// TIA Portal V19 export
FUNCTION_BLOCK "TYPIC_C402_IF_SBO1"   // FB111, FBD
TITLE = TYPIC_C402_IF_SBO: Afsluitboom
{ S7_Optimized_Access := 'TRUE' }
AUTHOR : OCOTECH
FAMILY : Typical
NAME : C402.704
// Logisch Object Besturing: C402.704
// 
// 								De interne functie afsluitboom verzorgt de interne besturing,
// 								bewaking en fysieke aansturing van een afsluitboom.
// 
// 								Het akoestisch signaal en de optische signalen behorend bij de
// 								afsluitboom, wordt eveneens via deze functie aangestuurd.
// stored: MemoryReserve 10, SetENOAutomatically false
   VAR_INPUT
      EXT_AUT { ExternalAccessible := 'False'; ExternalVisible := 'False'; ExternalWritable := 'False'} : Bool;   // Externe (hoofd) beveiliging (1 = OK)
      EXT_HW { ExternalAccessible := 'False'; ExternalVisible := 'False'; ExternalWritable := 'False'} : Bool;   // Sturings hardware (PLC) bewaking (1 = OK)
      HULP_KNIP { ExternalAccessible := 'False'; ExternalVisible := 'False'; ExternalWritable := 'False'} : Bool;   // Knippersignaal, x tijd hoog, x tijd laag
      IN_AUT { ExternalAccessible := 'False'; ExternalVisible := 'False'; ExternalWritable := 'False'} : Bool;   // Motorbeveiliging (1 = OK / 0 = storing)
      IN_OPEN { ExternalAccessible := 'False'; ExternalVisible := 'False'; ExternalWritable := 'False'} : Bool;   // Terugmelding: afsluitboom is open
      IN_TOE { ExternalAccessible := 'False'; ExternalVisible := 'False'; ExternalWritable := 'False'} : Bool;   // Terugmelding: afsluitboom is toe
      IN_STO { ExternalAccessible := 'False'; ExternalVisible := 'False'; ExternalWritable := 'False'} : Bool;   // Terugmelding: afsluitboom is buiten dienst
      IN_SCW { ExternalAccessible := 'False'; ExternalVisible := 'False'; ExternalWritable := 'False'} : Bool;   // Werkschakelaar (1 = AAN)
      IN_HND { ExternalAccessible := 'False'; ExternalVisible := 'False'; ExternalWritable := 'False'} : Bool;   // Mechanische handmatige bediening (0 = Hand)
      IN_LVE1_STO { ExternalAccessible := 'False'; ExternalVisible := 'False'; ExternalWritable := 'False'} : Bool;   // Detector lus 1 (1 = OK / 0 = storing)
      IN_LVE2_STO { ExternalAccessible := 'False'; ExternalVisible := 'False'; ExternalWritable := 'False'} : Bool;   // Detector lus 2 (1 = OK / 0 = storing)
      IN_LVE3_STO { ExternalAccessible := 'False'; ExternalVisible := 'False'; ExternalWritable := 'False'} : Bool;   // Detector lus 3 (1 = OK / 0 = storing)
      IN_LVE4_STO { ExternalAccessible := 'False'; ExternalVisible := 'False'; ExternalWritable := 'False'} : Bool;   // Detector lus 4 (1 = OK / 0 = storing)
      IN_LUS1_STS { ExternalAccessible := 'False'; ExternalVisible := 'False'; ExternalWritable := 'False'} : Bool;   // Detectie voertuig door lus 1 (1 = Geen detectie)
      IN_LUS2_STS { ExternalAccessible := 'False'; ExternalVisible := 'False'; ExternalWritable := 'False'} : Bool;   // Detectie voertuig door lus 2 (1 = Geen detectie)
      IN_LUS3_STS { ExternalAccessible := 'False'; ExternalVisible := 'False'; ExternalWritable := 'False'} : Bool;   // Detectie voertuig door lus 3 (1 = Geen detectie)
      IN_LUS4_STS { ExternalAccessible := 'False'; ExternalVisible := 'False'; ExternalWritable := 'False'} : Bool;   // Detectie voertuig door lus 4 (1 = Geen detectie)
      IN_AUT_C402 { ExternalAccessible := 'False'; ExternalVisible := 'False'; ExternalWritable := 'False'} : Bool;   // Beveiligingen: serie geschakelde terugmelding (1 = OK)
      IN_DKN_OPEN { ExternalAccessible := 'False'; ExternalVisible := 'False'; ExternalWritable := 'False'} : Bool;   // 1 = Drukknop ingedrukt, bediening openen
      IN_DKN_TOE { ExternalAccessible := 'False'; ExternalVisible := 'False'; ExternalWritable := 'False'} : Bool;   // 1 = Drukknop ingedrukt, bediening sluiten
      IN_DKN_STOP { ExternalAccessible := 'False'; ExternalVisible := 'False'; ExternalWritable := 'False'} : Bool;   // 1 = Drukknop ingedrukt, bediening stop
      CFG_TYD_STS { ExternalAccessible := 'False'; ExternalVisible := 'False'; ExternalWritable := 'False'} : Time;   // Vertragingstijd storing terugmelding stand bereikt
      CFG_ITYD_POS { ExternalAccessible := 'False'; ExternalVisible := 'False'; ExternalWritable := 'False'} : Time;   // Inschakelvertraging storing eindpositie terugmelding weggevallen
      CFG_UTYD_POS { ExternalAccessible := 'False'; ExternalVisible := 'False'; ExternalWritable := 'False'} : Time;   // Uitschakelvertraging storing eindpositie terugmelding weggevallen
      CFG_ITYD_OAS_SNEL { ExternalAccessible := 'False'; ExternalVisible := 'False'; ExternalWritable := 'False'} : Time;   // Vertragingstijd versneld sluiten afsluitboom na akoestisch en optisch signaal
      CFG_ITYD_OAS { ExternalAccessible := 'False'; ExternalVisible := 'False'; ExternalWritable := 'False'} : Time;   // Vertragingstijd sluiten/openen afsluitboom regulier na akoestisch en optisch signaal
      CFG_UTYD_OAS { ExternalAccessible := 'False'; ExternalVisible := 'False'; ExternalWritable := 'False'} : Time;   // Vertragingstijd uitschakelen akoestische en optische signalen
      CFG_UTYD_MOT { ExternalAccessible := 'False'; ExternalVisible := 'False'; ExternalWritable := 'False'} : Time;   // Vertragingstijd uitschakelen motor na bereiken eindpositie
      CFG_VGV_OPEN { ExternalAccessible := 'False'; ExternalVisible := 'False'; ExternalWritable := 'False'} : Bool;   // 1 = Slagboom moet openen bij bediening openen door hulpdiensten
   END_VAR
   VAR_OUTPUT
      VAR_IF_SBO { ExternalAccessible := 'False'; ExternalVisible := 'False'; ExternalWritable := 'False'} : "C402_VAR_IF_SBO_TYPIC";   // Struct met alle variabelen naar bovenliggende functies
      OUT_OPEN { ExternalAccessible := 'False'; ExternalVisible := 'False'; ExternalWritable := 'False'} : Bool;   // Aansturing openen
      OUT_TOE { ExternalAccessible := 'False'; ExternalVisible := 'False'; ExternalWritable := 'False'} : Bool;   // Aansturing sluiten
      OUT_AKS { ExternalAccessible := 'False'; ExternalVisible := 'False'; ExternalWritable := 'False'} : Bool;   // Aansturen akoestische signalering
      OUT_OPS { ExternalAccessible := 'False'; ExternalVisible := 'False'; ExternalWritable := 'False'} : Bool;   // Aansturen optische signalering
   END_VAR
   VAR_IN_OUT
      STU_IF_SBO : "C402_STU_IF_SBO_TYPIC";   // Struct met alle sturingen naar de functie (IF) in de interne sturing van de afsluitboom
      STU_AFS_IF_SBO : "C402_STU_AFS_IF_SBO_TYPIC";   // Struct met alle sturingen vanuit de interne functie Afsluitsysteem naar de functies (IF) van de afsluitbomen
   END_VAR
   VAR
      STO { ExternalWritable := 'False'} : Struct   // Storingen
         A001 { ExternalAccessible := 'False'; ExternalVisible := 'False'} : Bool;   // Beveiliging aangesproken
         A002 { ExternalAccessible := 'False'; ExternalVisible := 'False'} : Bool;   // Storing van de detector van lus 1
         A003 { ExternalAccessible := 'False'; ExternalVisible := 'False'} : Bool;   // Storing van de detector van lus 2
         A004 { ExternalAccessible := 'False'; ExternalVisible := 'False'} : Bool;   // Storing van de detector van lus 3
         A005 { ExternalAccessible := 'False'; ExternalVisible := 'False'} : Bool;   // Storing van de detector van lus 4
         A006 { ExternalAccessible := 'False'; ExternalVisible := 'False'} : Bool;   // Storing van de motorsturing
         A007 { ExternalAccessible := 'False'; ExternalVisible := 'False'} : Bool;   // Storing motorbeveiliging
         AT01 { ExternalAccessible := 'False'; ExternalVisible := 'False'} : Bool;   // Terugmelding Open niet tijdig bereikt
         AT02 { ExternalAccessible := 'False'; ExternalVisible := 'False'} : Bool;   // Terugmelding Dicht niet tijdig bereikt
         AT03 { ExternalAccessible := 'False'; ExternalVisible := 'False'} : Bool;   // Terugmeldingen Open en Dicht tegelijkertijd
         AT04 { ExternalAccessible := 'False'; ExternalVisible := 'False'} : Bool;   // Terugmelding Open weggevallen
         AT05 { ExternalAccessible := 'False'; ExternalVisible := 'False'} : Bool;   // Terugmelding Dicht weggevallen
         M001 { ExternalAccessible := 'False'; ExternalVisible := 'False'} : Bool;   // Werkschakelaar uitgeschakeld
         M002 { ExternalAccessible := 'False'; ExternalVisible := 'False'} : Bool;   // Mechanische handbediening uitgenomen
      END_STRUCT;
      VAR { ExternalWritable := 'False'} : Struct   // Variabelen
         CMD_AKS { ExternalAccessible := 'False'; ExternalVisible := 'False'} : Bool;   // Aansturen akoestische signalering
         CMD_OPS { ExternalAccessible := 'False'; ExternalVisible := 'False'} : Bool;   // Aansturen optische signalering
         VWA_AT04 { ExternalAccessible := 'False'; ExternalVisible := 'False'} : Bool;   // Voorwaarden voldaan voor storing AT04
         VWA_AT05 { ExternalAccessible := 'False'; ExternalVisible := 'False'} : Bool;   // Voorwaarden voldaan voor storing AT05
         MOT_STS_AAN { ExternalAccessible := 'False'; ExternalVisible := 'False'} : Bool;   // Motor afsluitboom aangestuurd
         CMD_OPEN { ExternalAccessible := 'False'; ExternalVisible := 'False'} : Bool;   // Gewenste stand afsluitboom is Open
         CMD_TOE { ExternalAccessible := 'False'; ExternalVisible := 'False'} : Bool;   // Gewenste stand afsluitboom is Toe
         CMD_STOP { ExternalAccessible := 'False'; ExternalVisible := 'False'} : Bool;   // Gewenste stand afsluitboom is Stop
         STO { ExternalAccessible := 'False'; ExternalVisible := 'False'} : Bool;   // De afsluitboom heeft een storing waardoor deze niet aangestuurd kan worden
         LOK_OPEN { ExternalAccessible := 'False'; ExternalVisible := 'False'} : Bool;   // Afsluitboom dient te openen voor hulpdiensten
         CMD_NEW { ExternalAccessible := 'False'; ExternalVisible := 'False'} : Bool;   // Nieuwe commando ontvangen vanuit 3B
         VGV_TOE { ExternalAccessible := 'False'; ExternalVisible := 'False'} : Bool;   // Vrijgave om de afsluitboom te sluiten
         CMD_TYD_OPEN { ExternalAccessible := 'False'; ExternalVisible := 'False'} : Bool;   // Gewenste stand afsluitboom is Open, tijdsvertraging OK
         CMD_TYD_TOE { ExternalAccessible := 'False'; ExternalVisible := 'False'} : Bool;   // Gewenste stand afsluitboom is Toe, tijdsvertraging OK
         STS_BEZ_OPEN { ExternalAccessible := 'False'; ExternalVisible := 'False'} : Bool;   // TRUE = Afsluitboom bezig met beweging openen
         STS_BEZ_TOE { ExternalAccessible := 'False'; ExternalVisible := 'False'} : Bool;   // TRUE = Afsluitboom bezig met beweging sluiten
         STS_OPEN { ExternalAccessible := 'False'; ExternalVisible := 'False'} : Bool;   // TRUE = Afsluitboom op stand Open
         STS_TOE { ExternalAccessible := 'False'; ExternalVisible := 'False'} : Bool;   // TRUE = Afsluitboom op stand Dicht
         STS_STOP { ExternalAccessible := 'False'; ExternalVisible := 'False'} : Bool;   // TRUE = Afsluitboom niet op een eindpositie en niet in beweging
         BMO_HAND { ExternalAccessible := 'False'; ExternalVisible := 'False'} : Bool;   // TRUE = Afsluitboom in hand geschakeld / FALSE = niet in hand
         STS_VKL_OK { ExternalAccessible := 'False'; ExternalVisible := 'False'} : Bool;   // TRUE = Verkeerslichten op Rood (voorwaarde voor sluiten)
         STS_NDS_OK { ExternalAccessible := 'False'; ExternalVisible := 'False'} : Bool;   // TRUE = Geen noodstop (voorwaarde voor beweging)
         STS_LUS_OK { ExternalAccessible := 'False'; ExternalVisible := 'False'} : Bool;   // TRUE = Detectielus(sen) OK (geen obstakel gedetecteerd voor sluiten)
         EXT_AUT { ExternalAccessible := 'False'; ExternalVisible := 'False'} : Bool;   // Externe (hoofd) beveiliging aangesproken
         EXT_HW { ExternalAccessible := 'False'; ExternalVisible := 'False'} : Bool;   // Sturings hardware (PLC) in storing
         EXT_STO { ExternalAccessible := 'False'; ExternalVisible := 'False'} : Bool;   // Externe storing aanwezig
         LUS1_STS { ExternalAccessible := 'False'; ExternalVisible := 'False'} : Bool;   // Detectie voertuig door lus 1 (1 = detectie)
         LUS2_STS { ExternalAccessible := 'False'; ExternalVisible := 'False'} : Bool;   // Detectie voertuig door lus 2 (1 = detectie)
         LUS3_STS { ExternalAccessible := 'False'; ExternalVisible := 'False'} : Bool;   // Detectie voertuig door lus 3 (1 = detectie)
         LUS4_STS { ExternalAccessible := 'False'; ExternalVisible := 'False'} : Bool;   // Detectie voertuig door lus 3 (1 = detectie)
      END_STRUCT;
   END_VAR
BEGIN

REGION Network 1: START
END_REGION

REGION Network 2: +++ Storingen en meldingen +++
   // Verwerken van de storingen en meldingen.
END_REGION

REGION Network 3: Storing A001: Beveiliging aangesproken
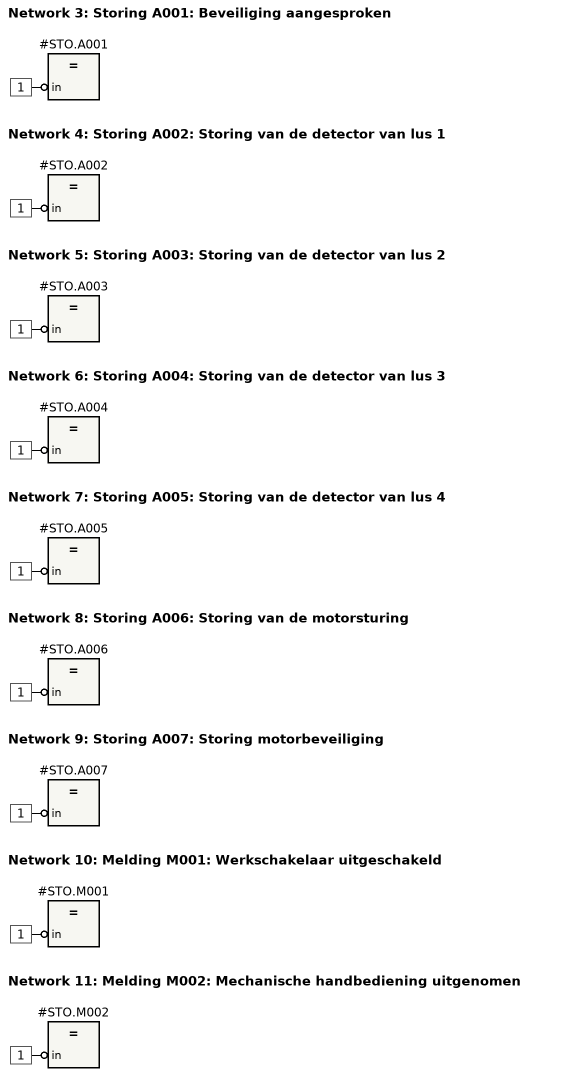
   #STO.A001 := NOT 1;
END_REGION

REGION Network 4: Storing A002: Storing van de detector van lus 1
   #STO.A002 := NOT 1;
END_REGION

REGION Network 5: Storing A003: Storing van de detector van lus 2
   #STO.A003 := NOT 1;
END_REGION

REGION Network 6: Storing A004: Storing van de detector van lus 3
   #STO.A004 := NOT 1;
END_REGION

REGION Network 7: Storing A005: Storing van de detector van lus 4
   #STO.A005 := NOT 1;
END_REGION

REGION Network 8: Storing A006: Storing van de motorsturing
   #STO.A006 := NOT 1;
END_REGION

REGION Network 9: Storing A007: Storing motorbeveiliging
   #STO.A007 := NOT 1;
END_REGION

REGION Network 10: Melding M001: Werkschakelaar uitgeschakeld
   #STO.M001 := NOT 1;
END_REGION

REGION Network 11: Melding M002: Mechanische handbediening uitgenomen
   #STO.M002 := NOT 1;
END_REGION

REGION Network 12: +++ Status detectielussen +++
   // De afsluitboom kan enkel voorwaardelijk sluiten als de
   // 										detectielussen geen metalen object detecteren en geen
   // 										storing hebben.
END_REGION

REGION Network 13: +++ Openen afsluitboom voor hulpdiensten +++
   // De afsluitboom kan door de hulpdiensten geopend worden als
   // 										op het bedieningspaneel de betreffende drukknop bediend
   // 										wordt en er vrijgave is voor bediening.
END_REGION

REGION Network 14: +++ Gewenste beweging afsluitboom +++
   // Afhankelijk van de werkingsmode, bedieningen en commandos
   // 										wordt de gewenste beweging van de afsluitboom bepaald
   // 										(openen / sluiten / stop).
END_REGION

REGION Network 15: +++ Vrijgave sluiten +++
   // Het sluiten van de afsluitboom mag enkel plaatsvinden als
   // 										er geen obstakel gedetecteerd wordt. Bij handbediening of
   // 										bij het commando onvoorwaardelijk sluiten wordt er geen
   // 										rekening gehouden met de obstakeldetectie.
END_REGION

REGION Network 16: +++ Tijdsvertraging aansturen afsluitboom +++
   // Vooraleer de afsluitboom aan te sturen, dienen de
   // 										akoestische en optische signalering aangestuurd te zijn. Pas
   // 										na een korte tijdsvertraging mag de afsluitboom in beweging
   // 										komen.
END_REGION

REGION Network 17: +++ Afsluitboomsturing +++
   // Aansturen van de afsluitboom en terugmeldingsbewaking.
END_REGION

REGION Network 18: +++ Sturing akoestische signalering +++
   // De akoestische signalering wordt aangestuurd van zodra de
   // 										afsluitboom dient te bewegen. De beweging wordt pas ingezet
   // 										nadat de akoestische signalering gedurende een bepaalde tijd
   // 										aangestuurd geweest is.
END_REGION

REGION Network 19: +++ Sturing Optische signalering +++
   // De optische signalering wordt aangestuurd van zodra de
   // 										afsluitboom dient te bewegen en blijft aangestuurd tot de
   // 										afsluitboom zich opnieuw in de open positie bevindt.
END_REGION

REGION Network 20 (SCL): EINDE
   // Variabelen van intern scada rakvlak naar outputs copieren
   #VAR_IF_SBO.STS_BEZ_OPEN := #VAR.STS_BEZ_OPEN;
   #VAR_IF_SBO.STS_BEZ_TOE := #VAR.STS_BEZ_TOE;
   #VAR_IF_SBO.STS_OPEN := #VAR.STS_OPEN;
   #VAR_IF_SBO.STS_TOE := #VAR.STS_TOE;
   #VAR_IF_SBO.STS_STOP := #VAR.STS_STOP;
   #VAR_IF_SBO.BMO_HAND := #VAR.BMO_HAND;
   #VAR_IF_SBO.STS_VKL_OK := #VAR.STS_VKL_OK;
   #VAR_IF_SBO.STS_NDS_OK := #VAR.STS_NDS_OK;
   #VAR_IF_SBO.STS_LUS_OK := #VAR.STS_LUS_OK;
   #VAR_IF_SBO.EXT_AUT := #VAR.EXT_AUT;
   #VAR_IF_SBO.EXT_HW := #VAR.EXT_HW;
   #VAR_IF_SBO.EXT_STO := #VAR.EXT_STO;
   #VAR_IF_SBO.LUS1_STS := #VAR.LUS1_STS;
   #VAR_IF_SBO.LUS2_STS := #VAR.LUS2_STS;
   #VAR_IF_SBO.LUS3_STS := #VAR.LUS3_STS;
   #VAR_IF_SBO.LUS4_STS := #VAR.LUS4_STS;
   #VAR_IF_SBO.STO := #STO;
END_REGION
END_FUNCTION_BLOCK
